// TIA Portal V17 export
// export: Created 2026-01-01T00:00:00, ExportSetting WithDefaults, DisplayName synthetic-fixture, DisplayVersion machine-intelligence-v1.0.0
FUNCTION_BLOCK "FB_Alarm"   // FB, SCL
BEGIN

NETWORK
TITLE = 
// network 1

NETWORK
TITLE = 
// network 2

NETWORK
TITLE = 
// network 3

NETWORK
TITLE = 
// network 4

NETWORK
TITLE = 
// network 5

NETWORK
TITLE = 
// network 6

NETWORK
TITLE = 
// network 7

NETWORK
TITLE = 
// network 8

NETWORK
TITLE = 
UNKNOWN_INSTRUCTION();
END_FUNCTION_BLOCK
